# EPICS substitutions: ecmcApp/Db/ecmcController.substitutions
file "ecmcController.template"
{
pattern
{P,      PORT, ADDR, TIMEOUT}
{IOC2:,  MCU1,    0, 1}
}
